{attribute addProperty BoxType "AX2000-B110-0000"}
{attribute addProperty Id "InputsAT %I*Inputs_352C0ED16480OutputsAT %Q*Outputs_39B5897F4860WcStateAT %I*WcState_98A4DF7520.250InfoDataAT %I*InfoData_6C7DEEF988110"}
{attribute addProperty CRC "4027785059"}
{attribute addProperty SizeInBites "202"}
{attribute addProperty SizeInBytes "25.25"}
TYPE AX2000_4A6B0158 :
STRUCT
	{attribute addProperty Name "Inputs"}
	Inputs : Inputs_352C0ED1;
	{attribute addProperty Name "Outputs"}
	Outputs : Outputs_39B5897F;
	{attribute addProperty Name "WcState"}
	WcState : WcState_98A4DF75;
	{attribute addProperty Name "InfoData"}
	InfoData : InfoData_6C7DEEF9;
END_STRUCT
END_TYPE

(* stored: Version 1.2.0.0, ProductVersion 3.1.4024.9
   DUT AX2000_4A6B0158: Id {a02c4537-d168-4bbc-a8e0-bc5c7876827c} *)
